// TIA Portal V20 export
DATA_BLOCK "IdentRfInterfaceHmi"   // DB218
// stored: InstanceOfName typeIdentRfHmi, InstanceOfType UDT
"typeIdentRfHmi"
   // VAR
   //    selectedUnit : USInt := 1;
   //    selectedEM : USInt;
   //    rfReaderId : USInt;
   //    numberOfRf : USInt;
   //    rfReader : Array[0.."NO_OF_RF_IDENT_DEVICES"] of "LSicar_typeIdentInterfaceHmi";
   // END_VAR
BEGIN
END_DATA_BLOCK
